// TIA Portal V20 export
FUNCTION "RealBlockName" : Void   // FC17, LAD
// Real block comment mentioning RealSite.
BEGIN

REGION Network 1
   // Real network comment.
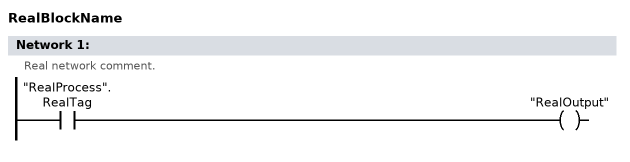
   RUNG wire#powerrail
      Contact( "RealProcess".RealTag )
      Coil( "RealOutput" )
   END_RUNG
   // the same network as SCL:
   "RealOutput" := "RealProcess".RealTag;
END_REGION
END_FUNCTION
